INTERFACE I_EtherCatMasterDiagnostic EXTENDS I_Component, I_Resettable

{attribute 'monitoring' := 'call'}
PROPERTY ConfiguredSlaveCount : UINT
GET
END_GET
END_PROPERTY

// Which subsystem produced ErrorId (see E_EcErrorSource for the meaning of ErrorId per source).
{attribute 'monitoring' := 'call'}
PROPERTY ErrorSource : E_EcErrorSource
GET
END_GET
END_PROPERTY

METHOD GetIoDeviceByAddr : I_EcIoDevice
VAR_INPUT
	Addr : WORD;
END_VAR
END_METHOD

METHOD GetIoDeviceByName : I_EcIoDevice
VAR_INPUT
	Name : STRING(31);
END_VAR
END_METHOD

// Configured slave index (0-based) of the slave with EtherCAT address Addr, -1 if none.
// O(1) for the dense address range starting at 1001, linear search otherwise.
METHOD GetSlaveIndexByAddr : DINT
VAR_INPUT
	Addr : UINT;
END_VAR
END_METHOD

{attribute 'monitoring' := 'call'}
PROPERTY LocalAmsNetId : T_AmsNetId
GET
END_GET
END_PROPERTY

{attribute 'monitoring' := 'call'}
PROPERTY MasterAmsNetId : T_AmsNetId
GET
END_GET
END_PROPERTY

METHOD RegisterEventProvider
VAR_INPUT
	EventProvider : I_EtherCatDiagnosticEventProvider;
END_VAR
END_METHOD

{attribute 'monitoring' := 'call'}
PROPERTY SlaveCount : UINT
GET
END_GET
END_PROPERTY

END_INTERFACE

(* stored: Version 1.1.0.1, ProductVersion 3.1.4026.18
   Itf I_EtherCatMasterDiagnostic: Id {d3244326-e8cc-4168-94a8-54382d32be09}
   Property ConfiguredSlaveCount: Id {96160ad3-3684-4597-872a-65dd5161395c}
   Get Get: Id {ffdd7ffe-1a36-4de4-bfc6-65ae3519bd6e}
   Property ErrorSource: Id {cf610482-1f30-43e7-aaf6-46b08c01425b}
   Get Get: Id {014fa14e-fe19-49d1-904f-1a044233a41a}
   Method GetIoDeviceByAddr: Id {32fe8214-5c95-4d51-ab86-b26ff0cba3b4}
   Method GetIoDeviceByName: Id {07e6d9ba-ce2c-4670-8bab-be3b592360a7}
   Method GetSlaveIndexByAddr: Id {7b3130f3-5ee6-4b64-b1f2-2e24132d8375}
   Property LocalAmsNetId: Id {632657fe-c107-0bc1-3a88-2ec0303b1452}
   Get Get: Id {f71aa313-7c5a-053b-17ba-71a4374885fd}
   Property MasterAmsNetId: Id {0844b1b5-8884-41ff-8311-005cb0130eaf}
   Get Get: Id {5d815bcb-9c01-4e07-92ac-c3e71960136a}
   Method RegisterEventProvider: Id {ab1390bb-ff23-4966-8077-63518787eb45}
   Property SlaveCount: Id {1e69259f-ee52-42e1-a0ed-fe5dbf856a8a}
   Get Get: Id {408a4639-9168-4575-b7b1-5a47bcabbee0} *)
